// TIA Portal V17 export
// export: Created 2025-04-25T10:07:24.9396604Z, ExportSetting WithDefaults, DisplayName Totally Integrated Automation Portal, DisplayVersion V17 Update 8, DisplayName TIA Portal Openness, DisplayVersion V17 Update 8, DisplayName TIA Portal Version Control Interface, DisplayVersion V17, DisplayName SINAMICS Startdrive Advanced, DisplayVersion V17 SP2, DisplayName SINAMICS Startdrive G110M, G120, G120C, G120D, G120P, G115D, DisplayVersion V17 SP2, DisplayName SINAMICS Startdrive G130, G150, S120, S150, SINAMICS MV, S210, DisplayVersion V17 SP2, DisplayName STEP 7 Professional, DisplayVersion V17 Update 8, DisplayName SINUMERIK ONE STEP 7 Toolbox, DisplayVersion V17 Update 12, DisplayName SINUMERIK 840D sl STEP 7 Toolbox, DisplayVersion V17 Update 12, DisplayName STEP 7 Safety, DisplayVersion V17 Update 6, DisplayName WinCC Advanced / Unified PC, DisplayVersion V17 Update 8
FUNCTION "FC2107_MACHINE_LIGHT" : Void   // FC2107, LAD
{ S7_Optimized_Access := 'FALSE' }
AUTHOR : ETXETAR
VERSION : 1.0
// stored: AutoNumber false, IsIECCheckEnabled false, SetENOAutomatically false, UDAEnableTagReadback false
BEGIN

REGION Network 1: MACHINE LIGHT
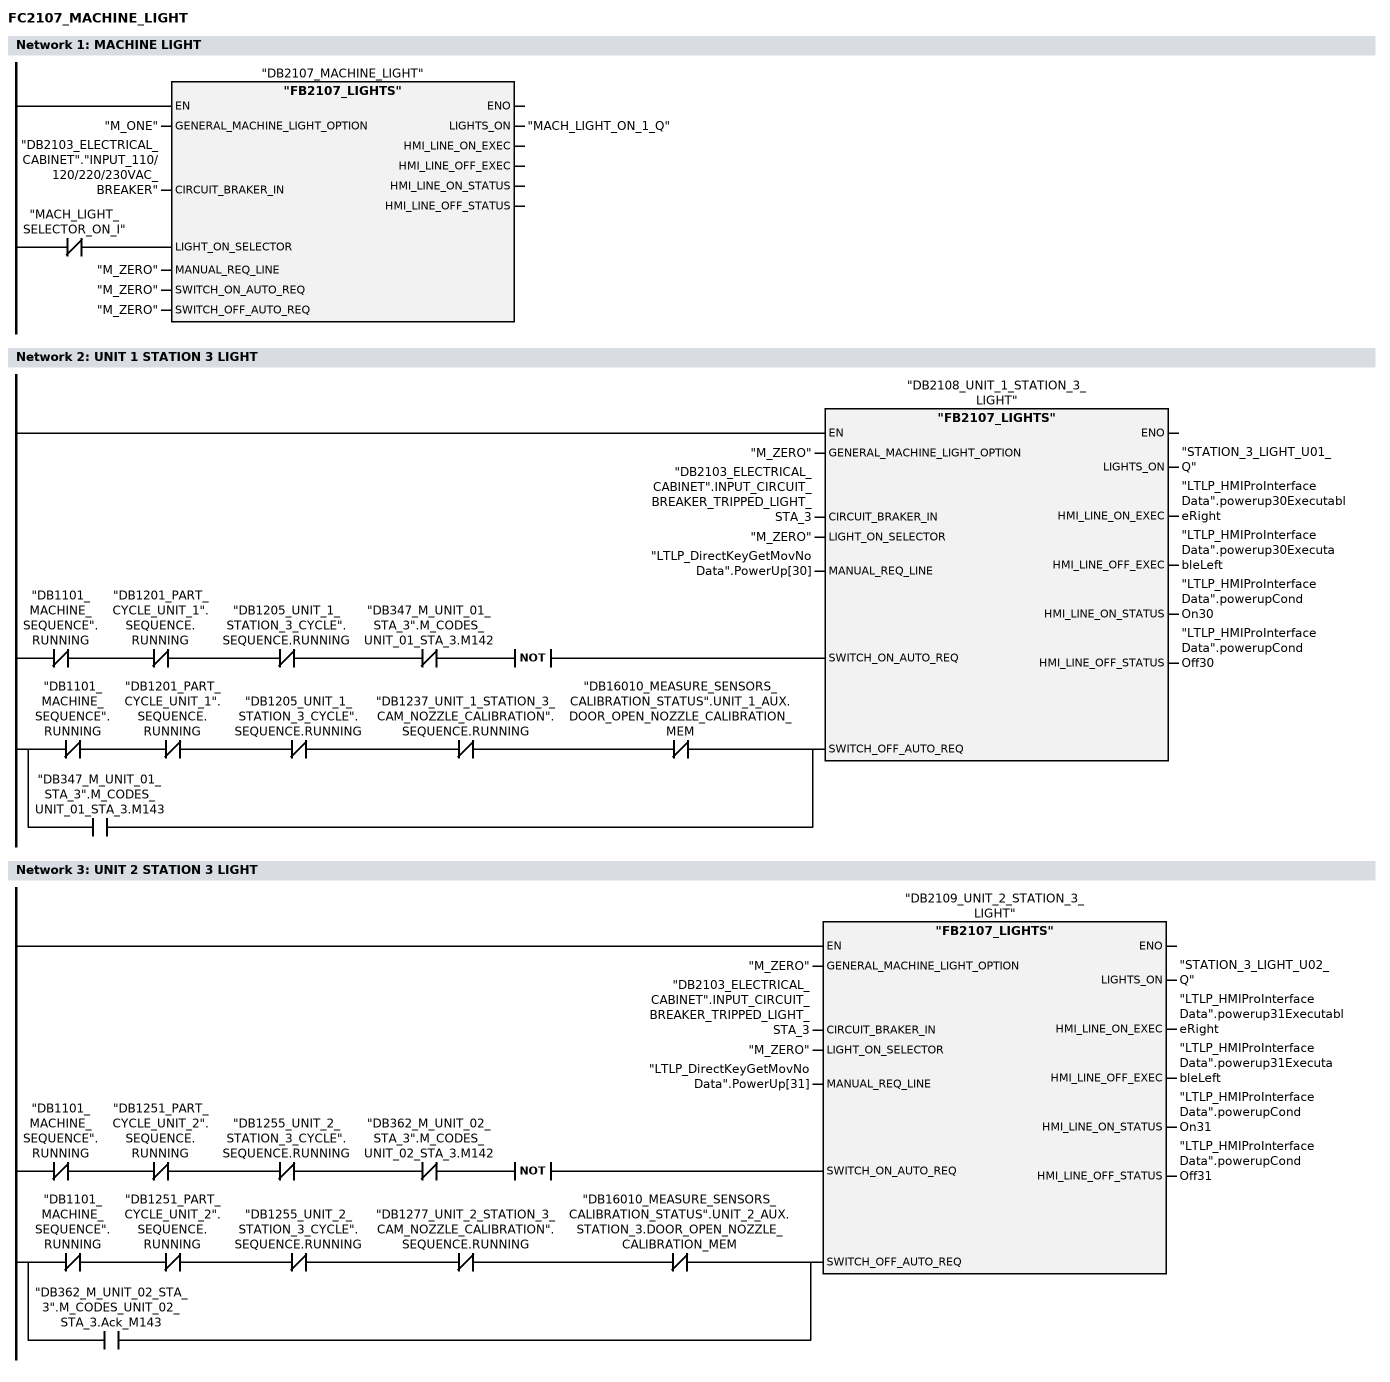
   RUNG wire#powerrail
      "DB2107_MACHINE_LIGHT"(LIGHT_ON_SELECTOR := wire#w1, GENERAL_MACHINE_LIGHT_OPTION := "M_ONE", CIRCUIT_BRAKER_IN := "DB2103_ELECTRICAL_CABINET"."INPUT_110/120/220/230VAC_BREAKER", MANUAL_REQ_LINE := "M_ZERO", SWITCH_ON_AUTO_REQ := "M_ZERO", SWITCH_OFF_AUTO_REQ := "M_ZERO", LIGHTS_ON => "MACH_LIGHT_ON_1_Q", HMI_LINE_ON_EXEC =>, HMI_LINE_OFF_EXEC =>, HMI_LINE_ON_STATUS =>, HMI_LINE_OFF_STATUS =>)
   END_RUNG
   RUNG wire#powerrail
      I_Contact( "MACH_LIGHT_SELECTOR_ON_I" )
   END_RUNG wire#w1
   // the same network as SCL:
   "DB2107_MACHINE_LIGHT"(GENERAL_MACHINE_LIGHT_OPTION := "M_ONE",   // "FB2107_LIGHTS"
                          CIRCUIT_BRAKER_IN := "DB2103_ELECTRICAL_CABINET"."INPUT_110/120/220/230VAC_BREAKER",
                          LIGHT_ON_SELECTOR := NOT "MACH_LIGHT_SELECTOR_ON_I",
                          MANUAL_REQ_LINE := "M_ZERO",
                          SWITCH_ON_AUTO_REQ := "M_ZERO",
                          SWITCH_OFF_AUTO_REQ := "M_ZERO",
                          LIGHTS_ON => "MACH_LIGHT_ON_1_Q");
END_REGION

REGION Network 2: UNIT 1 STATION 3 LIGHT
   RUNG wire#powerrail
      "DB2108_UNIT_1_STATION_3_LIGHT"(SWITCH_ON_AUTO_REQ := wire#w1, SWITCH_OFF_AUTO_REQ := wire#w2, GENERAL_MACHINE_LIGHT_OPTION := "M_ZERO", CIRCUIT_BRAKER_IN := "DB2103_ELECTRICAL_CABINET".INPUT_CIRCUIT_BREAKER_TRIPPED_LIGHT_STA_3, LIGHT_ON_SELECTOR := "M_ZERO", MANUAL_REQ_LINE := "LTLP_DirectKeyGetMovNoData".PowerUp[30], LIGHTS_ON => "STATION_3_LIGHT_U01_Q", HMI_LINE_ON_EXEC => "LTLP_HMIProInterfaceData".powerup30ExecutableRight, HMI_LINE_OFF_EXEC => "LTLP_HMIProInterfaceData".powerup30ExecutableLeft, HMI_LINE_ON_STATUS => "LTLP_HMIProInterfaceData".powerupCondOn30, HMI_LINE_OFF_STATUS => "LTLP_HMIProInterfaceData".powerupCondOff30)
   END_RUNG
   RUNG wire#powerrail
      I_Contact( "DB1101_MACHINE_SEQUENCE".RUNNING )
      I_Contact( "DB1201_PART_CYCLE_UNIT_1".SEQUENCE.RUNNING )
      I_Contact( "DB1205_UNIT_1_STATION_3_CYCLE".SEQUENCE.RUNNING )
      I_Contact( "DB347_M_UNIT_01_STA_3".M_CODES_UNIT_01_STA_3.M142 )
      Not()
   END_RUNG wire#w1
   RUNG wire#powerrail
      I_Contact( "DB1101_MACHINE_SEQUENCE".RUNNING )
      I_Contact( "DB1201_PART_CYCLE_UNIT_1".SEQUENCE.RUNNING )
      I_Contact( "DB1205_UNIT_1_STATION_3_CYCLE".SEQUENCE.RUNNING )
      I_Contact( "DB1237_UNIT_1_STATION_3_CAM_NOZZLE_CALIBRATION".SEQUENCE.RUNNING )
      I_Contact( "DB16010_MEASURE_SENSORS_CALIBRATION_STATUS".UNIT_1_AUX.DOOR_OPEN_NOZZLE_CALIBRATION_MEM )
   END_RUNG wire#w2
   RUNG wire#powerrail
      Contact( "DB347_M_UNIT_01_STA_3".M_CODES_UNIT_01_STA_3.M143 )
   END_RUNG wire#w2
   // the same network as SCL:
   "DB2108_UNIT_1_STATION_3_LIGHT"(GENERAL_MACHINE_LIGHT_OPTION := "M_ZERO",   // "FB2107_LIGHTS"
                           CIRCUIT_BRAKER_IN := "DB2103_ELECTRICAL_CABINET".INPUT_CIRCUIT_BREAKER_TRIPPED_LIGHT_STA_3,
                           LIGHT_ON_SELECTOR := "M_ZERO",
                           MANUAL_REQ_LINE := "LTLP_DirectKeyGetMovNoData".PowerUp[30],
                           SWITCH_ON_AUTO_REQ := NOT (NOT "DB1101_MACHINE_SEQUENCE".RUNNING AND NOT "DB1201_PART_CYCLE_UNIT_1".SEQUENCE.RUNNING AND NOT "DB1205_UNIT_1_STATION_3_CYCLE".SEQUENCE.RUNNING AND NOT "DB347_M_UNIT_01_STA_3".M_CODES_UNIT_01_STA_3.M142),
                           SWITCH_OFF_AUTO_REQ := (NOT "DB1101_MACHINE_SEQUENCE".RUNNING AND NOT "DB1201_PART_CYCLE_UNIT_1".SEQUENCE.RUNNING AND NOT "DB1205_UNIT_1_STATION_3_CYCLE".SEQUENCE.RUNNING AND NOT "DB1237_UNIT_1_STATION_3_CAM_NOZZLE_CALIBRATION".SEQUENCE.RUNNING AND NOT "DB16010_MEASURE_SENSORS_CALIBRATION_STATUS".UNIT_1_AUX.DOOR_OPEN_NOZZLE_CALIBRATION_MEM) OR "DB347_M_UNIT_01_STA_3".M_CODES_UNIT_01_STA_3.M143,
                           LIGHTS_ON => "STATION_3_LIGHT_U01_Q",
                           HMI_LINE_ON_EXEC => "LTLP_HMIProInterfaceData".powerup30ExecutableRight,
                           HMI_LINE_OFF_EXEC => "LTLP_HMIProInterfaceData".powerup30ExecutableLeft,
                           HMI_LINE_ON_STATUS => "LTLP_HMIProInterfaceData".powerupCondOn30,
                           HMI_LINE_OFF_STATUS => "LTLP_HMIProInterfaceData".powerupCondOff30);
END_REGION

REGION Network 3: UNIT 2 STATION 3 LIGHT
   RUNG wire#powerrail
      "DB2109_UNIT_2_STATION_3_LIGHT"(SWITCH_ON_AUTO_REQ := wire#w1, SWITCH_OFF_AUTO_REQ := wire#w2, GENERAL_MACHINE_LIGHT_OPTION := "M_ZERO", CIRCUIT_BRAKER_IN := "DB2103_ELECTRICAL_CABINET".INPUT_CIRCUIT_BREAKER_TRIPPED_LIGHT_STA_3, LIGHT_ON_SELECTOR := "M_ZERO", MANUAL_REQ_LINE := "LTLP_DirectKeyGetMovNoData".PowerUp[31], LIGHTS_ON => "STATION_3_LIGHT_U02_Q", HMI_LINE_ON_EXEC => "LTLP_HMIProInterfaceData".powerup31ExecutableRight, HMI_LINE_OFF_EXEC => "LTLP_HMIProInterfaceData".powerup31ExecutableLeft, HMI_LINE_ON_STATUS => "LTLP_HMIProInterfaceData".powerupCondOn31, HMI_LINE_OFF_STATUS => "LTLP_HMIProInterfaceData".powerupCondOff31)
   END_RUNG
   RUNG wire#powerrail
      I_Contact( "DB1101_MACHINE_SEQUENCE".RUNNING )
      I_Contact( "DB1251_PART_CYCLE_UNIT_2".SEQUENCE.RUNNING )
      I_Contact( "DB1255_UNIT_2_STATION_3_CYCLE".SEQUENCE.RUNNING )
      I_Contact( "DB362_M_UNIT_02_STA_3".M_CODES_UNIT_02_STA_3.M142 )
      Not()
   END_RUNG wire#w1
   RUNG wire#powerrail
      I_Contact( "DB1101_MACHINE_SEQUENCE".RUNNING )
      I_Contact( "DB1251_PART_CYCLE_UNIT_2".SEQUENCE.RUNNING )
      I_Contact( "DB1255_UNIT_2_STATION_3_CYCLE".SEQUENCE.RUNNING )
      I_Contact( "DB1277_UNIT_2_STATION_3_CAM_NOZZLE_CALIBRATION".SEQUENCE.RUNNING )
      I_Contact( "DB16010_MEASURE_SENSORS_CALIBRATION_STATUS".UNIT_2_AUX.STATION_3.DOOR_OPEN_NOZZLE_CALIBRATION_MEM )
   END_RUNG wire#w2
   RUNG wire#powerrail
      Contact( "DB362_M_UNIT_02_STA_3".M_CODES_UNIT_02_STA_3.Ack_M143 )
   END_RUNG wire#w2
   // the same network as SCL:
   "DB2109_UNIT_2_STATION_3_LIGHT"(GENERAL_MACHINE_LIGHT_OPTION := "M_ZERO",   // "FB2107_LIGHTS"
                           CIRCUIT_BRAKER_IN := "DB2103_ELECTRICAL_CABINET".INPUT_CIRCUIT_BREAKER_TRIPPED_LIGHT_STA_3,
                           LIGHT_ON_SELECTOR := "M_ZERO",
                           MANUAL_REQ_LINE := "LTLP_DirectKeyGetMovNoData".PowerUp[31],
                           SWITCH_ON_AUTO_REQ := NOT (NOT "DB1101_MACHINE_SEQUENCE".RUNNING AND NOT "DB1251_PART_CYCLE_UNIT_2".SEQUENCE.RUNNING AND NOT "DB1255_UNIT_2_STATION_3_CYCLE".SEQUENCE.RUNNING AND NOT "DB362_M_UNIT_02_STA_3".M_CODES_UNIT_02_STA_3.M142),
                           SWITCH_OFF_AUTO_REQ := (NOT "DB1101_MACHINE_SEQUENCE".RUNNING AND NOT "DB1251_PART_CYCLE_UNIT_2".SEQUENCE.RUNNING AND NOT "DB1255_UNIT_2_STATION_3_CYCLE".SEQUENCE.RUNNING AND NOT "DB1277_UNIT_2_STATION_3_CAM_NOZZLE_CALIBRATION".SEQUENCE.RUNNING AND NOT "DB16010_MEASURE_SENSORS_CALIBRATION_STATUS".UNIT_2_AUX.STATION_3.DOOR_OPEN_NOZZLE_CALIBRATION_MEM) OR "DB362_M_UNIT_02_STA_3".M_CODES_UNIT_02_STA_3.Ack_M143,
                           LIGHTS_ON => "STATION_3_LIGHT_U02_Q",
                           HMI_LINE_ON_EXEC => "LTLP_HMIProInterfaceData".powerup31ExecutableRight,
                           HMI_LINE_OFF_EXEC => "LTLP_HMIProInterfaceData".powerup31ExecutableLeft,
                           HMI_LINE_ON_STATUS => "LTLP_HMIProInterfaceData".powerupCondOn31,
                           HMI_LINE_OFF_STATUS => "LTLP_HMIProInterfaceData".powerupCondOff31);
END_REGION
END_FUNCTION
